(* CODESYS project Kicker.xml

Project tree, tasks and I/O mapping:
  function block Kicker [LD]
*)

// Kicker
FUNCTION_BLOCK Kicker
VAR_INPUT
	Enable: 			BOOL;
	Raise: 				BOOL;
	Lower: 				BOOL;
	Stop: 				BOOL;
	RaisedSensor: 		BOOL;
	LoweredSensor: 		BOOL;
END_VAR
VAR_OUTPUT
	Motor: 				BOOL;
	Brake: 				BOOL;
	Raised: 			BOOL;
	Lowered: 			BOOL;
END_VAR
VAR
	_RaiseTrigger: RS;
	_LowerTrigger: RS;
END_VAR
VAR // added by the converter: edge detectors and wires of the graphical bodies
    _w1 : BOOL;
    _rt1, _rt2 : R_TRIG;
END_VAR

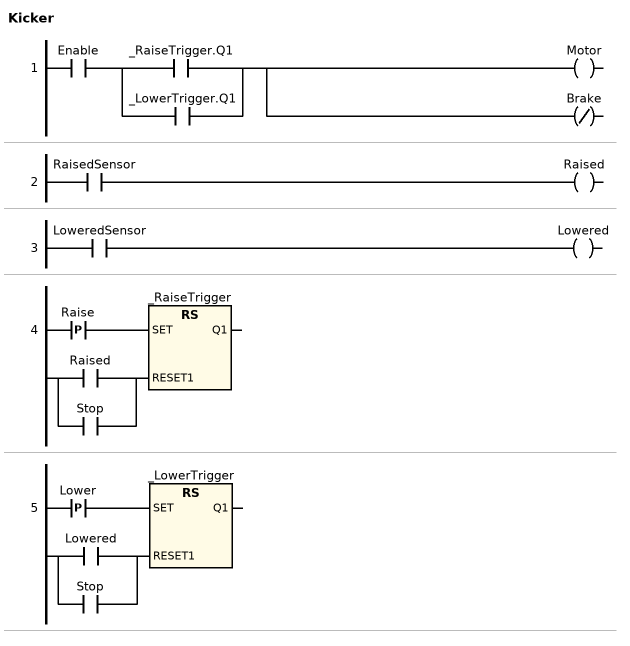
// NETWORK 1
_w1 := Enable AND (_RaiseTrigger.Q1 OR _LowerTrigger.Q1);
Motor := _w1;
Brake := NOT _w1;

// NETWORK 2
Raised := RaisedSensor;

// NETWORK 3
Lowered := LoweredSensor;

// NETWORK 4
_rt1(CLK := Raise);
_RaiseTrigger(SET := _rt1.Q, RESET1 := Raised OR Stop); // RS

// NETWORK 5
_rt2(CLK := Lower);
_LowerTrigger(SET := _rt2.Q, RESET1 := Lowered OR Stop); // RS

END_FUNCTION_BLOCK
